TYPE ST_P_GET_CHILD :
STRUCT
	Position:				INT;
	ContainerId:			INT;
	Barcode:				INT;
END_STRUCT
END_TYPE

(* stored: Version 1.1.0.1, ProductVersion 3.1.4024.10
   DUT ST_P_GET_CHILD: Id {a1b445f7-ebcc-4229-86ff-a94e2ba8a19e} *)
